ABB RAPID module: Module1.mod

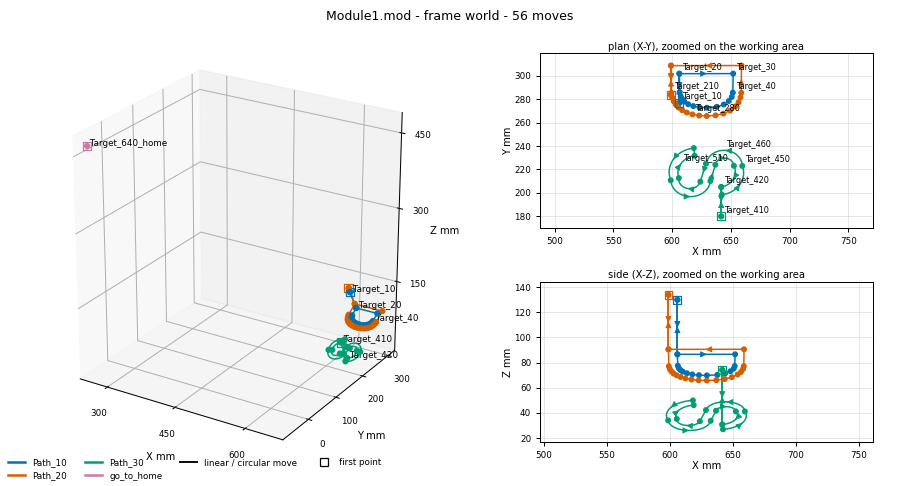
[picture p0: tool path of Module1.mod in frame world, 56 of 58 moves have a stored position in this frame; points joined in program order, loops and branches not executed]
MODULE Module1
        CONST robtarget Target_10:=[[-59.903986349,-18.467002478,65],[0,0.706526805,0.707686282,0],[0,0,0,0],[9E+09,9E+09,9E+09,9E+09,9E+09,9E+09]];
    CONST robtarget Target_20:=[[-59.903986349,-18.467002478,15],[0,0.706526805,0.707686282,0],[0,0,0,0],[9E+09,9E+09,9E+09,9E+09,9E+09,9E+09]];
    CONST robtarget Target_30:=[[-59.979150753,27.371954719,15],[0,0.706526805,0.707686282,0],[0,0,0,0],[9E+09,9E+09,9E+09,9E+09,9E+09,9E+09]];
    CONST robtarget Target_40:=[[-41.264483047,27.09568252,15],[0,0.706526805,0.707686282,0],[0,0,0,0],[9E+09,9E+09,9E+09,9E+09,9E+09,9E+09]];
    CONST robtarget Target_50:=[[-37.098585699,26.181639621,15],[0,0.706526805,0.707686282,0],[0,0,0,0],[9E+09,9E+09,9E+09,9E+09,9E+09,9E+09]];
    CONST robtarget Target_60:=[[-33.006751986,23.635483604,15],[0,0.706526805,0.707686282,0],[0,0,0,0],[9E+09,9E+09,9E+09,9E+09,9E+09,9E+09]];
    CONST robtarget Target_70:=[[-29.577255987,19.42042979,15],[0,0.706526805,0.707686282,0],[0,0,0,0],[9E+09,9E+09,9E+09,9E+09,9E+09,9E+09]];
    CONST robtarget Target_80:=[[-27.249655327,13.279967315,15],[0,0.706526805,0.707686282,0],[0,0,0,0],[9E+09,9E+09,9E+09,9E+09,9E+09,9E+09]];
    CONST robtarget Target_90:=[[-26.463498077,4.957575792,15],[0,0.706526805,0.707686282,0],[0,0,0,0],[9E+09,9E+09,9E+09,9E+09,9E+09,9E+09]];
    CONST robtarget Target_100:=[[-26.847117097,-1.33057448,15],[0,0.706526805,0.707686282,0],[0,0,0,0],[9E+09,9E+09,9E+09,9E+09,9E+09,9E+09]];
    CONST robtarget Target_110:=[[-28.020250242,-6.607063282,15],[0,0.706526805,0.707686282,0],[0,0,0,0],[9E+09,9E+09,9E+09,9E+09,9E+09,9E+09]];
    CONST robtarget Target_120:=[[-29.901014974,-10.89221746,15],[0,0.706526805,0.707686282,0],[0,0,0,0],[9E+09,9E+09,9E+09,9E+09,9E+09,9E+09]];
    CONST robtarget Target_130:=[[-32.407523991,-14.206359079,15],[0,0.706526805,0.707686282,0],[0,0,0,0],[9E+09,9E+09,9E+09,9E+09,9E+09,9E+09]];
    CONST robtarget Target_140:=[[-34.752828999,-15.990564546,15],[0,0.706526805,0.707686282,0],[0,0,0,0],[9E+09,9E+09,9E+09,9E+09,9E+09,9E+09]];
    CONST robtarget Target_150:=[[-37.784410563,-17.325684158,15],[0,0.706526805,0.707686282,0],[0,0,0,0],[9E+09,9E+09,9E+09,9E+09,9E+09,9E+09]];
    CONST robtarget Target_160:=[[-41.799075999,-18.161054214,15],[0,0.706526805,0.707686282,0],[0,0,0,0],[9E+09,9E+09,9E+09,9E+09,9E+09,9E+09]];
    CONST robtarget Target_170:=[[-59.903986349,-18.467002478,15],[0,0.706526805,0.707686282,0],[0,0,0,0],[9E+09,9E+09,9E+09,9E+09,9E+09,9E+09]];
    CONST robtarget Target_180:=[[-59.903986349,-18.467002478,65],[0,0.706526805,0.707686282,0],[0,0,0,0],[9E+09,9E+09,9E+09,9E+09,9E+09,9E+09]];
    CONST robtarget Target_190:=[[-67.832339525,-25.560505483,65],[0,0.706526805,0.707686282,0],[0,0,0,0],[9E+09,9E+09,9E+09,9E+09,9E+09,9E+09]];
    CONST robtarget Target_200:=[[-67.832339525,-25.560505483,15],[0,0.706526805,0.707686282,0],[0,0,0,0],[9E+09,9E+09,9E+09,9E+09,9E+09,9E+09]];
    CONST robtarget Target_210:=[[-41.050731723,-25.260795487,15],[0,0.706526805,0.707686282,0],[0,0,0,0],[9E+09,9E+09,9E+09,9E+09,9E+09,9E+09]];
    CONST robtarget Target_220:=[[-36.544835934,-24.486008035,15],[0,0.706526805,0.707686282,0],[0,0,0,0],[9E+09,9E+09,9E+09,9E+09,9E+09,9E+09]];
    CONST robtarget Target_230:=[[-32.658783027,-23.215991872,15],[0,0.706526805,0.707686282,0],[0,0,0,0],[9E+09,9E+09,9E+09,9E+09,9E+09,9E+09]];
    CONST robtarget Target_240:=[[-29.387431385,-21.466083208,15],[0,0.706526805,0.707686282,0],[0,0,0,0],[9E+09,9E+09,9E+09,9E+09,9E+09,9E+09]];
    CONST robtarget Target_250:=[[-26.541705712,-19.108069803,15],[0,0.706526805,0.707686282,0],[0,0,0,0],[9E+09,9E+09,9E+09,9E+09,9E+09,9E+09]];
    CONST robtarget Target_260:=[[-23.932516396,-16.013744164,15],[0,0.706526805,0.707686282,0],[0,0,0,0],[9E+09,9E+09,9E+09,9E+09,9E+09,9E+09]];
    CONST robtarget Target_270:=[[-21.667446852,-12.096312255,15],[0,0.706526805,0.707686282,0],[0,0,0,0],[9E+09,9E+09,9E+09,9E+09,9E+09,9E+09]];
    CONST robtarget Target_280:=[[-19.854080485,-7.268984806,15],[0,0.706526805,0.707686282,0],[0,0,0,0],[9E+09,9E+09,9E+09,9E+09,9E+09,9E+09]];
    CONST robtarget Target_290:=[[-18.666239149,-1.598541875,15],[0,0.706526805,0.707686282,0],[0,0,0,0],[9E+09,9E+09,9E+09,9E+09,9E+09,9E+09]];
    CONST robtarget Target_300:=[[-18.277768498,4.848212604,15],[0,0.706526805,0.707686282,0],[0,0,0,0],[9E+09,9E+09,9E+09,9E+09,9E+09,9E+09]];
    CONST robtarget Target_310:=[[-18.87852764,12.423979868,15],[0,0.706526805,0.707686282,0],[0,0,0,0],[9E+09,9E+09,9E+09,9E+09,9E+09,9E+09]];
    CONST robtarget Target_320:=[[-20.654497514,19.107640203,15],[0,0.706526805,0.707686282,0],[0,0,0,0],[9E+09,9E+09,9E+09,9E+09,9E+09,9E+09]];
    CONST robtarget Target_330:=[[-23.615721709,24.786626732,15],[0,0.706526805,0.707686282,0],[0,0,0,0],[9E+09,9E+09,9E+09,9E+09,9E+09,9E+09]];
    CONST robtarget Target_340:=[[-27.772253351,29.348372558,15],[0,0.706526805,0.707686282,0],[0,0,0,0],[9E+09,9E+09,9E+09,9E+09,9E+09,9E+09]];
    CONST robtarget Target_350:=[[-31.797703743,31.971378511,15],[0,0.706526805,0.707686282,0],[0,0,0,0],[9E+09,9E+09,9E+09,9E+09,9E+09,9E+09]];
    CONST robtarget Target_360:=[[-36.57874096,33.631342192,15],[0,0.706526805,0.707686282,0],[0,0,0,0],[9E+09,9E+09,9E+09,9E+09,9E+09,9E+09]];
    CONST robtarget Target_370:=[[-41.092068546,34.268555836,15],[0,0.706526805,0.707686282,0],[0,0,0,0],[9E+09,9E+09,9E+09,9E+09,9E+09,9E+09]];
    CONST robtarget Target_380:=[[-67.930724367,34.439418622,15],[0,0.706526805,0.707686282,0],[0,0,0,0],[9E+09,9E+09,9E+09,9E+09,9E+09,9E+09]];
    CONST robtarget Target_390:=[[-67.832339525,-25.560505483,15],[0,0.706526805,0.707686282,0],[0,0,0,0],[9E+09,9E+09,9E+09,9E+09,9E+09,9E+09]];
    CONST robtarget Target_400:=[[-67.832339525,-25.560505483,65],[0,0.706526805,0.707686282,0],[0,0,0,0],[9E+09,9E+09,9E+09,9E+09,9E+09,9E+09]];
    CONST robtarget Target_410:=[[51.565720132,17.159209824,65],[0,0.706526805,0.707686282,0],[0,0,0,0],[9E+09,9E+09,9E+09,9E+09,9E+09,9E+09]];
    CONST robtarget Target_420:=[[51.565720132,17.159209824,15],[0,0.706526805,0.707686282,0],[0,0,0,0],[9E+09,9E+09,9E+09,9E+09,9E+09,9E+09]];
    CONST robtarget Target_430:=[[59.17732298,17.744683087,15],[0,0.706526805,0.707686282,0],[0,0,0,0],[9E+09,9E+09,9E+09,9E+09,9E+09,9E+09]];
    CONST robtarget Target_440:=[[48.367011814,33.504604134,15],[0,0.706526805,0.707686282,0],[0,0,0,0],[9E+09,9E+09,9E+09,9E+09,9E+09,9E+09]];
    CONST robtarget Target_450:=[[30.816600488,35.112936384,15],[0,0.706526805,0.707686282,0],[0,0,0,0],[9E+09,9E+09,9E+09,9E+09,9E+09,9E+09]];
    CONST robtarget Target_460:=[[15.505237169,19.064613253,15],[0,0.706526805,0.707686282,0],[0,0,0,0],[9E+09,9E+09,9E+09,9E+09,9E+09,9E+09]];
    CONST robtarget Target_470:=[[28.595773923,4.213955722,15],[0,0.706526805,0.707686282,0],[0,0,0,0],[9E+09,9E+09,9E+09,9E+09,9E+09,9E+09]];
    CONST robtarget Target_480:=[[46.315178904,-0.612041693,15],[0,0.706526805,0.707686282,0],[0,0,0,0],[9E+09,9E+09,9E+09,9E+09,9E+09,9E+09]];
    CONST robtarget Target_490:=[[52.948382403,-11.748860171,15],[0,0.706526805,0.707686282,0],[0,0,0,0],[9E+09,9E+09,9E+09,9E+09,9E+09,9E+09]];
    CONST robtarget Target_500:=[[42.764052131,-18.943265798,15],[0,0.706526805,0.707686282,0],[0,0,0,0],[9E+09,9E+09,9E+09,9E+09,9E+09,9E+09]];
    CONST robtarget Target_510:=[[29.276034509,-17.522681396,15],[0,0.706526805,0.707686282,0],[0,0,0,0],[9E+09,9E+09,9E+09,9E+09,9E+09,9E+09]];
    CONST robtarget Target_520:=[[20.74331749,-5.483448358,15],[0,0.706526805,0.707686282,0],[0,0,0,0],[9E+09,9E+09,9E+09,9E+09,9E+09,9E+09]];
    CONST robtarget Target_530:=[[13.254634258,-6.150569272,15],[0,0.706526805,0.707686282,0],[0,0,0,0],[9E+09,9E+09,9E+09,9E+09,9E+09,9E+09]];
    CONST robtarget Target_540:=[[25.214440428,-24.057317621,15],[0,0.706526805,0.707686282,0],[0,0,0,0],[9E+09,9E+09,9E+09,9E+09,9E+09,9E+09]];
    CONST robtarget Target_550:=[[44.970063385,-25.810399574,15],[0,0.706526805,0.707686282,0],[0,0,0,0],[9E+09,9E+09,9E+09,9E+09,9E+09,9E+09]];
    CONST robtarget Target_560:=[[61.021018218,-8.405130388,15],[0,0.706526805,0.707686282,0],[0,0,0,0],[9E+09,9E+09,9E+09,9E+09,9E+09,9E+09]];
    CONST robtarget Target_570:=[[45.6410996,7.997027296,15],[0,0.706526805,0.707686282,0],[0,0,0,0],[9E+09,9E+09,9E+09,9E+09,9E+09,9E+09]];
    CONST robtarget Target_580:=[[29.641719798,12.186350796,15],[0,0.706526805,0.707686282,0],[0,0,0,0],[9E+09,9E+09,9E+09,9E+09,9E+09,9E+09]];
    CONST robtarget Target_590:=[[23.15783878,19.609221987,15],[0,0.706526805,0.707686282,0],[0,0,0,0],[9E+09,9E+09,9E+09,9E+09,9E+09,9E+09]];
    CONST robtarget Target_600:=[[30.710655582,27.965753216,15],[0,0.706526805,0.707686282,0],[0,0,0,0],[9E+09,9E+09,9E+09,9E+09,9E+09,9E+09]];
    CONST robtarget Target_610:=[[43.009513289,27.919410925,15],[0,0.706526805,0.707686282,0],[0,0,0,0],[9E+09,9E+09,9E+09,9E+09,9E+09,9E+09]];
    CONST robtarget Target_620:=[[51.565720132,17.159209824,15],[0,0.706526805,0.707686282,0],[0,0,0,0],[9E+09,9E+09,9E+09,9E+09,9E+09,9E+09]];
    CONST robtarget Target_630:=[[51.565720132,17.159209824,65],[0,0.706526805,0.707686282,0],[0,0,0,0],[9E+09,9E+09,9E+09,9E+09,9E+09,9E+09]];
    CONST robtarget Target_640_home:=[[257.237,-71.213623454,468.933097512],[0.39255433,-0.605404549,0.624448253,0.299083283],[0,-1,-1,0],[9E+09,9E+09,9E+09,9E+09,9E+09,9E+09]];
        TASK PERS tooldata tool1:=[TRUE,[[0,0,0],[1,0,0,0]],[-1,[0,0,0],[1,0,0,0],0,0,0]];
    CONST robtarget Target_640:=[[553.364448405,0,452.545222089],[0.489061793,0.013465943,0.869637173,-0.066094009],[0,-1,0,0],[9E+09,9E+09,9E+09,9E+09,9E+09,9E+09]];
    CONST jointtarget JointHome:=[[0,0,0,0,0,0],[9E+09,9E+09,9E+09,9E+09,9E+09,9E+09]];
    CONST jointtarget JointTarget_3:=[[4.353448171,17.58168898,18.597879402,1.064855093,26.739405892,-18.332137232],[9E+09,9E+09,9E+09,9E+09,9E+09,9E+09]];
!***********************************************************
    !
    ! Module:  Module1
    !
    ! Description:
    !   <Insert description here>
    !
    ! Author: jhair
    !
    ! Version: 1.0
    !
    !***********************************************************


    !***********************************************************
    !
    ! Procedure main
    !
    !   This is the entry point of your program
    !
    !***********************************************************
    PROC main()
        !Add your code here
        return_home;
        medium_point;
        Path_10;
        Path_20;
        Path_30;
        medium_point;
        return_home;
    ENDPROC
    PROC Path_10()
        MoveL Target_10,v200,fine,ToolM_DS109\WObj:=initials_wo0209;
        MoveL Target_20,v200,fine,ToolM_DS109\WObj:=initials_wo0209;
        MoveL Target_30,v200,fine,ToolM_DS109\WObj:=initials_wo0209;
        MoveL Target_40,v200,fine,ToolM_DS109\WObj:=initials_wo0209;
        MoveL Target_50,v200,fine,ToolM_DS109\WObj:=initials_wo0209;
        MoveL Target_60,v200,fine,ToolM_DS109\WObj:=initials_wo0209;
        MoveL Target_70,v200,fine,ToolM_DS109\WObj:=initials_wo0209;
        MoveL Target_80,v200,fine,ToolM_DS109\WObj:=initials_wo0209;
        MoveL Target_90,v200,fine,ToolM_DS109\WObj:=initials_wo0209;
        MoveL Target_100,v200,fine,ToolM_DS109\WObj:=initials_wo0209;
        MoveL Target_110,v200,fine,ToolM_DS109\WObj:=initials_wo0209;
        MoveL Target_120,v200,fine,ToolM_DS109\WObj:=initials_wo0209;
        MoveL Target_130,v200,fine,ToolM_DS109\WObj:=initials_wo0209;
        MoveL Target_140,v200,fine,ToolM_DS109\WObj:=initials_wo0209;
        MoveL Target_150,v200,fine,ToolM_DS109\WObj:=initials_wo0209;
        MoveL Target_160,v200,fine,ToolM_DS109\WObj:=initials_wo0209;
        MoveL Target_170,v200,fine,ToolM_DS109\WObj:=initials_wo0209;
        MoveL Target_180,v200,fine,ToolM_DS109\WObj:=initials_wo0209;
    ENDPROC
    PROC Path_20()
        MoveL Target_190,v200,fine,ToolM_DS109\WObj:=initials_wo0209;
        MoveL Target_200,v200,fine,ToolM_DS109\WObj:=initials_wo0209;
        MoveL Target_210,v200,fine,ToolM_DS109\WObj:=initials_wo0209;
        MoveL Target_220,v200,fine,ToolM_DS109\WObj:=initials_wo0209;
        MoveL Target_230,v200,fine,ToolM_DS109\WObj:=initials_wo0209;
        MoveL Target_240,v200,fine,ToolM_DS109\WObj:=initials_wo0209;
        MoveL Target_250,v200,fine,ToolM_DS109\WObj:=initials_wo0209;
        MoveL Target_260,v200,fine,ToolM_DS109\WObj:=initials_wo0209;
        MoveL Target_270,v200,fine,ToolM_DS109\WObj:=initials_wo0209;
        MoveL Target_280,v200,fine,ToolM_DS109\WObj:=initials_wo0209;
        MoveL Target_290,v200,fine,ToolM_DS109\WObj:=initials_wo0209;
        MoveL Target_300,v200,fine,ToolM_DS109\WObj:=initials_wo0209;
        MoveL Target_310,v200,fine,ToolM_DS109\WObj:=initials_wo0209;
        MoveL Target_320,v200,fine,ToolM_DS109\WObj:=initials_wo0209;
        MoveL Target_330,v200,fine,ToolM_DS109\WObj:=initials_wo0209;
        MoveL Target_340,v200,fine,ToolM_DS109\WObj:=initials_wo0209;
        MoveL Target_350,v200,fine,ToolM_DS109\WObj:=initials_wo0209;
        MoveL Target_360,v200,fine,ToolM_DS109\WObj:=initials_wo0209;
        MoveL Target_370,v200,fine,ToolM_DS109\WObj:=initials_wo0209;
        MoveL Target_380,v200,fine,ToolM_DS109\WObj:=initials_wo0209;
        MoveL Target_390,v200,fine,ToolM_DS109\WObj:=initials_wo0209;
        MoveL Target_400,v200,fine,ToolM_DS109\WObj:=initials_wo0209;
    ENDPROC
    PROC Path_30()
        MoveL Target_410,v200,fine,ToolM_DS109\WObj:=initials_wo0209;
        MoveL Target_420,v200,fine,ToolM_DS109\WObj:=initials_wo0209;
        MoveL Target_430,v200,fine,ToolM_DS109\WObj:=initials_wo0209;
        MoveC Target_440,Target_450,v200,fine,ToolM_DS109\WObj:=initials_wo0209;
        MoveC Target_460,Target_470,v200,fine,ToolM_DS109\WObj:=initials_wo0209;
        MoveL Target_480,v200,fine,ToolM_DS109\WObj:=initials_wo0209;
        MoveC Target_490,Target_500,v200,fine,ToolM_DS109\WObj:=initials_wo0209;
        MoveC Target_510,Target_520,v200,fine,ToolM_DS109\WObj:=initials_wo0209;
        MoveL Target_530,v200,fine,ToolM_DS109\WObj:=initials_wo0209;
        MoveC Target_540,Target_550,v200,fine,ToolM_DS109\WObj:=initials_wo0209;
        MoveC Target_560,Target_570,v200,fine,ToolM_DS109\WObj:=initials_wo0209;
        MoveL Target_580,v200,fine,ToolM_DS109\WObj:=initials_wo0209;
        MoveC Target_590,Target_600,v200,fine,ToolM_DS109\WObj:=initials_wo0209;
        MoveC Target_610,Target_620,v200,fine,ToolM_DS109\WObj:=initials_wo0209;
        MoveL Target_630,v200,fine,ToolM_DS109\WObj:=initials_wo0209;
    ENDPROC
    PROC go_to_home()
        MoveL Target_640_home,v1000,z100,ToolM_DS109\WObj:=wobj0;
    ENDPROC
    PROC return_home()
        MoveAbsJ JointHome,v1000,z100,ToolM_DS109\WObj:=initials_wo0209;
    ENDPROC
    PROC medium_point()
        MoveAbsJ JointTarget_3,v1000,z100,ToolM_DS109\WObj:=initials_wo0209;
    ENDPROC
ENDMODULE
